Fanuc KAREL source: kt00550.KL

-- PROVISIONAL review KL for V940-1; original PC SHA256 a69f992b1cf1271af30fc07143f0608795937a8c240cec2a5c9b5d685bf64296
-- Incomplete behavior may be omitted. Consult companion uncertainty JSON. Do not deploy.
PROGRAM KT00550
%NOLOCKGROUP
-- UNRESOLVED_DECL P1 type=000199
-- UNRESOLVED_DECL P2 type=000199
-- UNRESOLVED_DECL OUT type=000102
BEGIN
  -- V9_ZERO_TABLE_METADATA_HINT layout=0001; no indexed target words; source/name/runtime held
  -- UNRESOLVED_PC offsets 5-44; opcodes 49,7E,49,7E,60,7E,4A
  -- UNRESOLVED_PC offsets 49-53; opcodes 7F
END KT00550
